FUNCTION CEILING : LREAL
VAR_INPUT
	in : LREAL;
END_VAR

IF in - TRUNC(in) > 0 THEN
	CEILING := TRUNC(in) + 1;
ELSE
	CEILING := in;
END_IF

END_FUNCTION

(* stored: Version 1.1.0.1, ProductVersion 3.1.4024.11
   POU CEILING: Id {be585c52-13bc-4d17-a95c-9a2d812699f1}, SpecialFunc None *)
